Staubli VAL3: printLog.pgx

public program printLog(string x_sMessage)
  local num i
  local num l_nSize
begin
  // check the size after is 200 clear it and keep the first 50
  setMutex(bLogMutex)
  // do it
  if size(sLog)>=200
    // clean it
    delete(sLog[0])
  endIf
  // add one
  if sLog!=""
    insert(sLog[size(sLog)])
  endIf
  // write it
  sLog[size(sLog)-1]=x_sMessage
  //release
  bLogMutex=false
end
